// TIA Portal V17 export
// export: Created 2025-11-19T10:30:00.000Z, ExportSetting WithDefaults, DisplayName Totally Integrated Automation Portal, DisplayVersion V17
ORGANIZATION_BLOCK "Main"   // OB1, LAD, ProgramCycle
{ S7_Optimized_Access := 'TRUE' }
VERSION : 0.1
// stored: AutoNumber true, IsIECCheckEnabled false
   VAR_INPUT
      Initial_Call : Bool;
      Remanence : Bool;
   END_VAR
BEGIN

REGION Network 1: Motor Control Logic
   // Start motor when button pressed
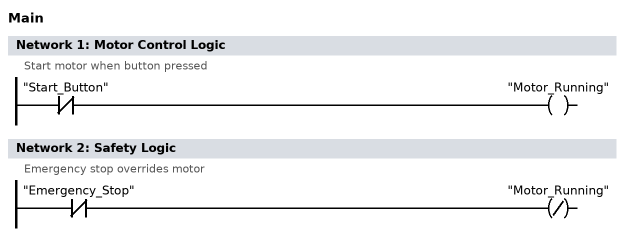
   RUNG wire#powerrail
      I_Contact( "Start_Button" )
      Coil( "Motor_Running" )
   END_RUNG
   // the same network as SCL:
   "Motor_Running" := NOT "Start_Button";
END_REGION

REGION Network 2: Safety Logic
   // Emergency stop overrides motor
   RUNG wire#powerrail
      I_Contact( "Emergency_Stop" )
      I_Coil( "Motor_Running" )
   END_RUNG
   // the same network as SCL:
   "Motor_Running" := NOT (NOT "Emergency_Stop");
END_REGION
END_ORGANIZATION_BLOCK
